Universal Robots PolyScope program: 6_wash_loop.urp

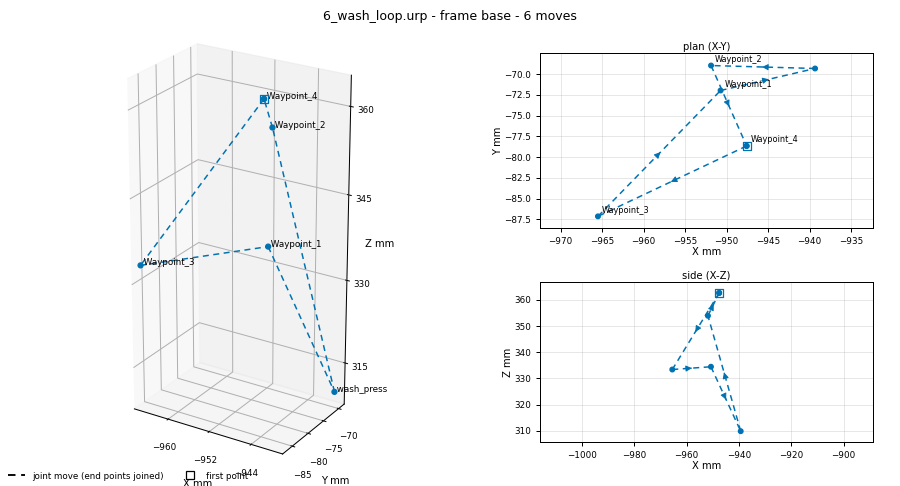
[picture p0: tool path of 6_wash_loop.urp in frame base, 6 of 6 moves have a stored position in this frame; points joined in program order, loops and branches not executed]
Program 6_wash_loop (installation=default directory=/programs/washer_rahman createdIn=5.9.5.1031259 lastSavedIn=5.9.5.1031259 robotSerialNumber=20215500597)
Calibrated DH parameters: a=[0.000193, -0.066673, -0.391568, -0.000012, 0.00005, 0]; d=[0.162643, -472.05677, 465.132521, 7.058239, 0.099746, 0.099582]; alpha=[1.571116, 0.00089, 0.003862, 1.569269, -1.569248, 0]; deltaTheta=[0, -1.413394, 7.628392, 0.068187, 0, -0.000001]
Robot Program (runOnlyOnce=true)
  SuppressedNode
    var_2 := 2
  SuppressedNode
    Script: glass_hover=p[-.200,-0.23+var_2*0.150 ,0.377,2.067,2.652,-2.043]
  SuppressedNode
    Script: glass_hover=p[-.603,-0.23+GP_int_in[0]*0.150 ,0.377,2.067,2.652,-2.043]
  MoveJ speed 60 deg/s, acceleration 80 deg/s^2 (useActiveTCP=true) feature=Base
    Waypoint Waypoint_4: TCP in base x=-947.575 y=-78.658 z=362.695 mm, rx=-1.3566 ry=-1.4371 rz=0.8681 rad; joints [-2.083, -50.768, 70.998, -182.431, -94.109, -8.128] deg; TCP offset x=0 y=0 z=191.5 mm, rx=0 ry=0 rz=0 rad
    Waypoint Waypoint_3: TCP in base x=-965.491 y=-87.139 z=333.412 mm, rx=-1.3367 ry=-1.4136 rz=1.0288 rad; joints [-3.622, -46.183, 70.562, -190.288, -87.254, -4.408] deg
    Waypoint Waypoint_1: TCP in base x=-950.716 y=-71.972 z=334.473 mm, rx=-1.3479 ry=-1.4172 rz=0.9935 rad; joints [-4.45, -48.651, 74.003, -190.275, -87.742, -5.317] deg
    Waypoint wash_press: TCP in base x=-939.332 y=-69.323 z=309.83 mm, rx=-1.3577 ry=-1.4049 rz=0.9729 rad; joints [-4.2, -48.472, 77.577, -193.86, -89.249, -5.297] deg
    Wait Sleep waitTime=5
  MoveJ speed 60 deg/s, acceleration 80 deg/s^2 (useActiveTCP=true) feature=Base
    Waypoint Waypoint_2: TCP in base x=-951.863 y=-68.965 z=353.967 mm, rx=-1.3447 ry=-1.3256 rz=0.9789 rad; joints [-3.135, -48.016, 72.481, -192.566, -92.591, -4.136] deg
    Waypoint Waypoint_4: TCP in base x=-947.575 y=-78.658 z=362.695 mm, rx=-1.3566 ry=-1.4371 rz=0.8681 rad; joints [-2.083, -50.768, 70.998, -182.431, -94.109, -8.128] deg
